FUNCTION_BLOCK CM_DigOutput EXTENDS CM_Base

VAR CONSTANT
	c_MAX_FB_NAME_LENGTH : USINT := 8; //Maximum feedback-name length
END_VAR

VAR_INPUT
	i_stSettings : ST_DigOutputSettings;
	i_bIclkOn : BOOL := TRUE; //TRUE = interlocked
	i_bIclkOff : BOOL := TRUE; //TRUE = interlocked
	
	i_ref_eCtrlState : REFERENCE TO E_CtrlState;
END_VAR

VAR
	// Outputs
	Q_bStaOutput AT %Q* : BOOL;
	
	// Force outputs (IO-test functions)
	s_fbForceCmdOutput : FB_ForceOutput;
	
	// Interlocks
	s_sInterlockedReasonOn : STRING(GVL.g_MAX_LEN_INTERLOCK_REASON); //External interlocked reason for clarifying reason
	s_sInterlockedReasonOff : STRING(GVL.g_MAX_LEN_INTERLOCK_REASON); //External interlocked reason for clarifying reason
	s_wrnOnInterlocked : BOOL;
	s_wrnOffInterlocked : BOOL;
	
	// Request
	s_bReqOff : BOOL;
	s_bReqOn : BOOL;
	
	// Status
	s_bStaOutputIsOff : BOOL;
	s_bStaOutputIsOn : BOOL;
	s_bStaWarning : BOOL;
	
	{attribute 'hide'}
	s_bStaOutput			: BOOL;
	
	{attribute: 'Hide'}
	s_bCfgReverseOutput : BOOL; // FALSE = NORMAL, TRUE = INVERTED
	
	s_sCfgOffName : STRING(c_MAX_FB_NAME_LENGTH) := 'Off';
	s_sCfgOnName : STRING(c_MAX_FB_NAME_LENGTH) := 'On';
	
	// Alarms
	// none

	// Hmi
	stHmiData : ST_DigOutput_HMI;
	
	s_fbHmiBtnManualOff		: FB_HmiBtn;
	s_fbHmiBtnManualOn		: FB_HmiBtn;
	
	s_fbHmiLedIsOff			: FB_HmiLed;
	s_fbHmiLedIsOn			: FB_HmiLed;

END_VAR


m_Main();

METHOD PROTECTED _m_Hmi : BOOL

IF NOT SUPER^._m_Hmi() THEN
	RETURN;
END_IF

//To Hmi
stHmiData.sDescription := i_sCmName;
stHmiData.sNameOff := s_fbHmiBtnManualOff.p_sBtnText;
stHmiData.sNameOn := s_fbHmiBtnManualOn.p_sBtnText;
stHmiData.bStaOff := NOT(s_bStaOutput);
stHmiData.bStaOn := s_bStaOutput;
stHmiData.bBtnOffEnabled := s_fbHmiBtnManualOff.p_bStaEnabled;
stHmiData.bBtnOnEnabled := s_fbHmiBtnManualOn.p_bStaEnabled;
stHmiData.s_sInterlockedReason := s_sInterlockedReasonOn;

//From Hmi
IF stHmiData.bCmdOffPressed THEN
	s_fbHmiBtnManualOff.m_On();
ELSE
	s_fbHmiBtnManualOff.m_Off();	
END_IF

IF stHmiData.bCmdOnPressed THEN
	s_fbHmiBtnManualOn.m_On();
ELSE
	s_fbHmiBtnManualOn.m_Off();	
END_IF 

//Buttons
s_fbHmiBtnManualOff();
s_fbHmiBtnManualOn();

//Led
s_fbHmiLedIsOff(i_bStaLed := NOT(s_bStaOutput));
s_fbHmiLedIsOn(i_bStaLed := s_bStaOutput);
		
IF __ISVALIDREF(i_ref_eCtrlState) THEN
	//MAINTENANCE-mode is running
	IF (i_eCtrlMode = E_CtrlMode.MAINTENANCE) AND (i_ref_eCtrlState = E_CtrlState.RUNNING) THEN
		s_fbHmiBtnManualOff.p_bStaVisible := TRUE;
		s_fbHmiBtnManualOff.p_bStaEnabled := i_bReqEnable AND NOT(i_bIclkOff);
		
		s_fbHmiBtnManualOn.p_bStaVisible := TRUE;
		s_fbHmiBtnManualOn.p_bStaEnabled := i_bReqEnable AND NOT(i_bIclkOn);
			
		IF s_fbHmiBtnManualOff.p_osrBtnPress THEN
			m_Off();
		END_IF
			
		IF s_fbHmiBtnManualOn.p_osrBtnPress THEN
			m_On();
		END_IF
		
	//other-mode	
	ELSE
		s_fbHmiBtnManualOff.p_bStaVisible := FALSE;
		s_fbHmiBtnManualOff.p_bStaEnabled := FALSE;
	
		s_fbHmiBtnManualOn.p_bStaVisible := FALSE;
		s_fbHmiBtnManualOn.p_bStaEnabled := FALSE;

		s_fbHmiBtnManualOn.p_bStaVisible := FALSE;
		s_fbHmiBtnManualOn.p_bStaEnabled := FALSE;
	END_IF
END_IF	
	
_m_Hmi := TRUE;
END_METHOD

METHOD PROTECTED _m_Init : BOOL

IF NOT SUPER^._m_Init() THEN
	RETURN;
END_IF

//Hmi 
	s_fbHmiBtnManualOff.p_eButtontype := E_HmiButtonType.PUSHBUTTON;
	s_fbHmiBtnManualOff.p_bStaVisible := FALSE;
	s_fbHmiBtnManualOff.p_bStaEnabled := FALSE;		
	s_fbHmiBtnManualOff.p_sBtnText := s_sCfgOffName;
	
	s_fbHmiBtnManualOn.p_eButtontype := E_HmiButtonType.PUSHBUTTON;
	s_fbHmiBtnManualon.p_bStaVisible := FALSE;
	s_fbHmiBtnManualOn.p_bStaEnabled := FALSE;		
	s_fbHmiBtnManualon.p_sBtnText := s_sCfgOnName;
	
	s_fbHmiLedIsOff.p_bStaVisible := FALSE;
	s_fbHmiLedIsOff.p_sToHmiDescriptionLed := CONCAT('Is at: ', s_sCfgOffName);
	
	s_fbHmiLedIsOn.p_bStaVisible := FALSE;
	s_fbHmiLedIsOn.p_sToHmiDescriptionLed := CONCAT('Is at: ', s_sCfgOnName);

_m_Init := TRUE;
END_METHOD

METHOD PROTECTED _m_Outputs : BOOL
VAR_INST
	s_bCmdOutput : BOOL;
END_VAR

IF NOT SUPER^._m_Outputs() THEN
	RETURN;
END_IF

IF i_bReqEnable AND s_bReqOff AND NOT(i_bIclkOff) THEN
			s_bCmdOutput := FALSE;
		ELSIF i_bReqEnable AND s_bReqOn AND NOT(i_bIclkOn) THEN
			s_bCmdOutput := TRUE;
		ELSE
			s_bCmdOutput := FALSE;	
		END_IF

IF __ISVALIDREF(i_ref_eCtrlState) THEN
	IF (i_eCtrlMode <> E_CtrlMode.IO) OR (i_ref_eCtrlState <> E_CtrlState.RUNNING) THEN
		s_fbForceCmdOutput.i_eForceValue := E_ForceValue.RELEASED; 	
	END_IF
END_IF
	
s_fbForceCmdOutput(
	i_ref_bCmdInput := s_bCmdOutput,
	i_ref_bCmdOutput := Q_bStaOutput);

_m_Outputs := TRUE;
END_METHOD

METHOD PUBLIC m_Main : BOOL

s_bStaOutput := i_bStaOutput;

IF NOT s_bInitDone THEN
	IF _m_Init() THEN
		s_bInitDone := TRUE;
	END_IF 
END_IF

s_osrOn(CLK := s_bStaOutput);
s_osfOff(CLK := s_bStaOutput);

s_tonDelay(IN := s_bStaOutput <> s_bStaOutputDelayed, PT := i_stSettings.tmOutputDelay);

IF s_bStaOutput AND s_tonDelay.Q THEN
	s_bStaOutputDelayed := TRUE;
END_IF

IF NOT s_bStaOutput AND s_tonDelay.Q THEN
	s_bStaOutputDelayed := FALSE;
END_IF

_m_Outputs();

m_Main := TRUE;
END_METHOD

METHOD PUBLIC m_Off : BOOL

IF NOT i_bReqEnable THEN 
	RETURN;
END_IF

IF NOT(i_bIclkOff) THEN
	s_bReqOff := TRUE XOR s_bCfgReverseOutput;
	s_bReqOn := FALSE XOR s_bCfgReverseOutput;
ELSE
	s_wrnOffInterlocked := TRUE;
END_IF	
	
m_off := s_bStaOutputIsOff;
END_METHOD

METHOD PUBLIC m_On : BOOL

IF NOT i_bReqEnable THEN 
	RETURN;
END_IF

IF NOT(i_bIclkOn) THEN
	s_bReqOff := FALSE XOR s_bCfgReverseOutput;
	s_bReqOn := TRUE XOR s_bCfgReverseOutput;
ELSE
	s_wrnOnInterlocked := TRUE;
END_IF
	
m_On := s_bStaOutputIsOn;
END_METHOD

{attribute 'monitoring':='call'}
PROPERTY PUBLIC p_bCfgReverseOutput : BOOL
GET

p_bCfgReverseOutput := s_bCfgReverseOutput;
END_GET
SET

s_bCfgReverseOutput := p_bCfgReverseOutput;
END_SET
END_PROPERTY

{attribute 'monitoring':='call'}
PROPERTY PUBLIC p_bStaIsOff : BOOL
GET

p_bStaIsOff := s_bStaOutputIsOff;
END_GET
END_PROPERTY

{attribute 'monitoring':='call'}
PROPERTY PUBLIC p_bStaIsOn : BOOL
GET

p_bStaIsOn := s_bStaOutputIsOn;
END_GET
END_PROPERTY

{attribute 'monitoring':='call'}
PROPERTY PUBLIC p_bStaOutput : BOOL
GET
p_bStaOutput := s_bStaOutput;
END_GET
END_PROPERTY

{attribute 'monitoring':='call'}
PROPERTY PUBLIC p_bStaWarning : BOOL
GET

p_bStaWarning := s_bStaWarning;
END_GET
END_PROPERTY

{attribute 'monitoring':='call'}
PROPERTY PUBLIC p_sCfgOffName : STRING(c_MAX_FB_NAME_LENGTH)
GET

p_sCfgOffName := s_sCfgOffName;
END_GET
SET

s_sCfgOffName := p_sCfgOffName;
END_SET
END_PROPERTY

{attribute 'monitoring':='call'}
PROPERTY PUBLIC p_sCfgOnName : STRING(c_MAX_FB_NAME_LENGTH)
GET

p_sCfgOnName := s_sCfgOnName;
END_GET
SET

s_sCfgOnName := p_sCfgOnName;
END_SET
END_PROPERTY

{attribute 'monitoring':='call'}
PROPERTY PUBLIC p_sInterlockedReasonOff : STRING(GVL.g_MAX_LEN_INTERLOCK_REASON)
GET

p_sInterlockedReasonOff := s_sInterlockedReasonOff;
END_GET
SET

s_sInterlockedReasonOff := p_sInterlockedReasonOff;
END_SET
END_PROPERTY

{attribute 'monitoring':='call'}
PROPERTY PUBLIC p_sInterlockedReasonOn : STRING(GVL.g_MAX_LEN_INTERLOCK_REASON)
GET

p_sInterlockedReasonOn := s_sInterlockedReasonOn;
END_GET
SET

s_sInterlockedReasonOn := p_sInterlockedReasonOn;
END_SET
END_PROPERTY

END_FUNCTION_BLOCK

(* stored: Version 1.1.0.1, ProductVersion 3.1.4024.12
   POU CM_DigOutput: Id {f6926334-60a3-431a-8319-95017baa0ee2}, SpecialFunc None
   Folder Methods: Id {8e6d06cb-4405-49f8-902f-b0c016a886d0}
   Folder Properties: Id {445cfafc-a5c1-4426-9164-91ffc9a267f4}
   Method _m_Hmi: Id {f4e34c00-dde3-49d5-b728-851a846aadfb}
   Method _m_Init: Id {58eaf209-c641-4c2f-b3df-64ebcea68410}
   Method _m_Outputs: Id {e570ab94-2a26-4b08-93d9-96af8fab708a}
   Method m_Main: Id {2dd33bfc-7121-4f83-aa70-6c1522573289}
   Method m_Off: Id {ecec5de6-8993-4f02-85de-c763a17adf6c}
   Method m_On: Id {72dee1e9-15f6-4acf-a222-f05c7a0f3b2a}
   Property p_bCfgReverseOutput: Id {91faff52-ccfa-4828-8537-1e596812f30f}
   Get Get: Id {36007a3c-1d2d-4d74-b650-7e1855152a36}
   Set Set: Id {dad35811-9b82-45a9-b984-ddbbd50110e7}
   Property p_bStaIsOff: Id {b7c83b24-d0ae-42f1-a82a-ab2f516b13a1}
   Get Get: Id {5dec523d-3816-4f0a-bd4f-cf74110f9c1d}
   Property p_bStaIsOn: Id {a5094957-1772-4d40-9c14-e5eba61eb945}
   Get Get: Id {aa06a3e2-4e28-4410-9202-80b549a4969f}
   Property p_bStaOutput: Id {cdc0ff34-12d0-4b48-b5e8-b09853bb5cc9}
   Get Get: Id {42e85b44-18f0-412a-9346-64d13e29ff2a}
   Property p_bStaWarning: Id {3d0e8e10-0192-43a6-a918-fca531311cfd}
   Get Get: Id {1864105f-9395-4c47-afc3-a0e6285c2bde}
   Property p_sCfgOffName: Id {bad7f86a-ed76-4fc4-b545-49766b502d8b}
   Get Get: Id {ecdac295-9e12-42e1-af6a-1438fc907ace}
   Set Set: Id {cc069142-38c9-413b-93f9-16c3e3887d0b}
   Property p_sCfgOnName: Id {c262eae1-1891-4a87-a7b5-82eb7fd3a41c}
   Get Get: Id {f4a2f70f-caa9-4957-9aec-eceee385e016}
   Set Set: Id {a5550812-774b-4113-93cf-353687427523}
   Property p_sInterlockedReasonOff: Id {34e39de3-1002-4b2d-9f20-9e3d7e031852}
   Get Get: Id {02af5916-8462-404d-ba13-c9bf19efff4c}
   Set Set: Id {63c7fba6-aadc-432b-8f62-3e22ecb87594}
   Property p_sInterlockedReasonOn: Id {9f60b92c-c8a8-4ac7-9e39-6da66771e2a7}
   Get Get: Id {92330fa5-6f16-48b5-8c4f-5e514f368ece}
   Set Set: Id {ed995ebe-f73e-4698-bbee-a8437daca919} *)
